// SIMATIC S7-200 SMART project (STEP 7-Micro/WIN SMART), CPU ST40

ORGANIZATION_BLOCK MAIN:OB1
TITLE=Program Comments
BEGIN
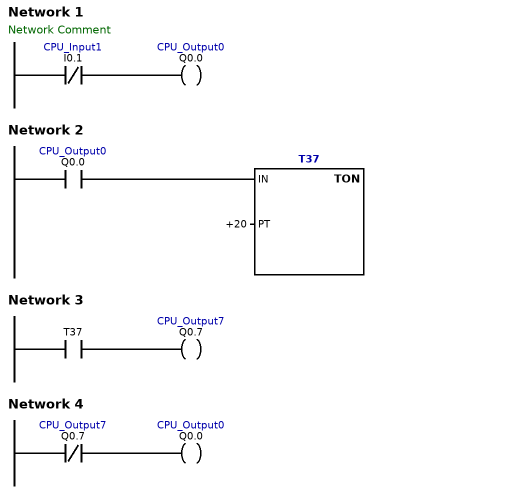
Network 1
// Network Comment
LDN    CPU_Input1:I0.1
=      CPU_Output0:Q0.0
Network 2
LD     CPU_Output0:Q0.0
TON    T37, +20
Network 3
LD     T37
=      CPU_Output7:Q0.7
Network 4
LDN    CPU_Output7:Q0.7
=      CPU_Output0:Q0.0
END_ORGANIZATION_BLOCK
